// TIA Portal V21 export
TYPE "Std_StatoUtenza"
   STRUCT
      Stato : Int;
      K : Int;   // Valore della costante
      ValoreAttuale : "Std_ValoreConUm";   // Posizione / analogica attuale / velocità
   END_STRUCT;
END_TYPE
